FUNCTION_BLOCK U_MAIN
VAR_INPUT
END_VAR
VAR_OUTPUT
END_VAR
VAR
	initDone	: BOOL;
	typeshift	: U_typeshift;
END_VAR

IF NOT initDone THEN
	Cfg();
	initDone := TRUE;	
END_IF

//calls
typeshift();

END_FUNCTION_BLOCK

(* stored: Version 1.1.0.1
   POU U_MAIN: Id {f64e1143-92d9-4aba-8f2a-567bdd906705}, SpecialFunc None *)
